PROGRAM Fixture1_Auto
VAR
	
nState_Door    : INT; // 0: Idle, 10: Starting, 20: Rotating, 30: Stopping
	
END_VAR




/////////////// OPERATOR LOAD PART FIX 1 ///////////////

		IF Memory_DB.M_Auto_Active AND 
		   Memory_DB.M_Power_On AND 
		   Inputs.i_Front_Door_Up
		   THEN   
		IF Memory_DB.M_FX1_LOAD1 AND Memory_DB.M_Turntable_POS1_Reached AND Memory_DB.M_Fixture1_TR_POS1_Reached  THEN
		  Inputs.i_FX1_PART_CONTROL_B1 := TRUE;
		  Inputs.i_FX1_PART_CONTROL_B2 := TRUE;
		  Inputs.i_FX1_PART_CONTROL_B3 := TRUE;
		  Inputs.i_FX1_PART_CONTROL_B4 := TRUE;
		  Inputs.i_FX1_PART_CONTROL_B5 := TRUE;
		  Inputs.i_FX1_PART_CONTROL_B6 := TRUE;
		  Inputs.i_FX1_PART_CONTROL_B7 := TRUE;
		  Memory_DB.M_FX1_LOAD1_COMPLETED :=TRUE;
		
		ELSIF Memory_DB.M_Auto_Active AND Memory_DB.M_Turntable_POS1_Reached AND Memory_DB.M_Fixture1_TR_POS2_Reached AND Memory_DB.M_FX1_LOAD2 THEN
		      Inputs.i_FX1_PART_CONTROL_B15 := TRUE;
		      Inputs.i_FX1_PART_CONTROL_B16 := TRUE;
		      Inputs.i_FX1_PART_CONTROL_B17 := TRUE;
		      Inputs.i_FX1_PART_CONTROL_B18 := TRUE;
		      Inputs.i_FX1_PART_CONTROL_B19 := TRUE;
		      Inputs.i_FX1_PART_CONTROL_B20 := TRUE;
		      Inputs.i_FX1_PART_CONTROL_B21 := TRUE;
		      Memory_DB.M_FX1_LOAD2_COMPLETED :=TRUE;
		
		ELSIF Memory_DB.M_FX1_LOAD1_COMPLETED AND Memory_DB.M_FX1_LOAD2_COMPLETED THEN
			
			  Memory_DB.M_Fixture1_TR_Start :=TRUE;
			
		END_IF;
		END_IF;
		 IF 
		   Memory_DB. M_FX1_All_Initialise THEN
		   Memory_DB.M_Turntable_Start := TRUE;
	       Memory_DB.M_Turntable_POS1_CMD := TRUE;
		   Memory_DB.M_Turntable_POS2_CMD := FALSE;
		   Memory_DB.M_Fixture1_TR_Start := TRUE;
	       Memory_DB.M_Fixture1_TR_POS1_CMD := TRUE;
		   Memory_DB.M_Fixture1_TR_POS2_CMD := FALSE;
		   Memory_DB.M_REAR_DOOR_DOWN := TRUE;
		   Memory_DB.M_REAR_DOOR_Up := FALSE;
		   
		 END_IF
//////////////////LODING SIDE DOOR & TRUNION CONTROL OPERATION/////////////////
IF  Memory_DB.M_Auto_Active AND Memory_DB.M_Safety_Ok AND Memory_DB.M_Power_On  THEN
	
CASE nState_Door  OF
    0: // Default Position1 of Door Open
	IF Memory_DB.M_Turntable_POS1_Reached AND Memory_DB.M_Fixture1_TR_POS1_Reached THEN      
		Memory_DB.M_FRONT_DOOR_Down	:=FALSE;
		Memory_DB.M_FRONT_DOOR_UP	:=TRUE;	
		Memory_DB.M_R03_MH_Goto_Drop2:=FALSE;
		nState_Door := 10;
     END_IF  
	 
    10: // 1st Load completed and Door Close Command
 
        IF Memory_DB.M_FX1_LOAD1_COMPLETED AND Memory_DB.M_FX1_Cycle_Start_PB AND Inputs.i_Front_Door_Up THEN
		Memory_DB.M_FRONT_DOOR_Down	:=TRUE;
		Memory_DB.M_FRONT_DOOR_UP	:=FALSE;

            nState_Door := 20; // Trunion Move
        END_IF
		       
    20: // Clamp Sequence at Trunion Pos1
 
        IF Inputs.i_Front_Door_Down AND Memory_DB.M_Fixture1_TR_POS1_Reached THEN
		Memory_DB.A_FX1_CC1_CLAMPING_UNIT1_3_WP:=TRUE;
		Memory_DB.A_FX1_CC3_CLAMPING_UNIT3_3_WP:=TRUE;
		Memory_DB.A_FX1_CC5_CLAMPING_UNIT5_1_WP:=TRUE;
		Memory_DB.A_FX1_CC1_CLAMPING_UNIT1_3_HP:=FALSE;
		Memory_DB.A_FX1_CC3_CLAMPING_UNIT3_3_HP:=FALSE;
		Memory_DB.A_FX1_CC5_CLAMPING_UNIT5_1_HP:=FALSE;		

         nState_Door := 30; // Error State
        END_IF	

        
    30: // Trunion move to Position 2 for 2nd Load
 
        IF Inputs.i_Front_Door_Down AND Inputs.i_FX1_CC1_Clamp_1_Sensor_WP AND 
		Inputs.i_FX1_CC3_Clamp_1_Sensor_WP AND Inputs.i_FX1_CC5_Clamp_1_Sensor_WP THEN
		Memory_DB.M_Fixture1_TR_POS2_CMD:=TRUE;
		Memory_DB.M_Fixture1_TR_POS1_CMD:=FALSE;

            nState_Door := 40; // Error State
        END_IF		
        
    40: // Door Open command for 2nd Load
 
        IF Memory_DB.M_Fixture1_TR_POS2_Reached AND Inputs.i_Front_Door_Down THEN
		Memory_DB.M_FRONT_DOOR_Down:=FALSE;
		Memory_DB.M_FRONT_DOOR_UP  :=TRUE;

            nState_Door := 50; // Error State
        END_IF	
        
    50: // 2nd Load completed on Trunion & Door Close Command
 
        IF Memory_DB.M_FX1_LOAD2_COMPLETED AND Memory_DB.M_FX1_Cycle_Start_PB AND Inputs.i_Front_Door_Up THEN
		Memory_DB.M_FRONT_DOOR_Down      :=TRUE;
		Memory_DB.M_FRONT_DOOR_Up        :=FALSE;

            nState_Door := 60; // Error State
        END_IF
		
    60: // Clamp Sequence at Trunion Pos1
 
        IF Inputs.i_Front_Door_Down AND Memory_DB.M_Fixture1_TR_POS2_Reached THEN
		Memory_DB.A_FX1_CC2_CLAMPING_UNIT2_3_WP:=TRUE;
		Memory_DB.A_FX1_CC4_CLAMPING_UNIT4_3_WP:=TRUE;
		Memory_DB.A_FX1_CC6_CLAMPING_UNIT6_1_WP:=TRUE;
		Memory_DB.A_FX1_CC2_CLAMPING_UNIT2_3_HP:=FALSE;
		Memory_DB.A_FX1_CC4_CLAMPING_UNIT4_3_HP:=FALSE;
		Memory_DB.A_FX1_CC6_CLAMPING_UNIT6_1_HP:=FALSE;	

         nState_Door := 70; // Error State
        END_IF		
        
    70: // Move Trunion to Default/Pos1
 
        IF Memory_DB.M_Fixture1_TR_Start AND Inputs.i_Front_Door_Down AND Memory_DB.M_Fixture1_TR_POS2_Reached AND
		 Inputs.i_FX1_CC2_Clamp_1_Sensor_WP AND Inputs.i_FX1_CC4_Clamp_1_Sensor_WP AND Inputs.i_FX1_CC6_Clamp_1_Sensor_WP THEN
		Memory_DB.M_Fixture1_TR_POS1_CMD:=TRUE;
		Memory_DB.M_Fixture1_TR_POS2_CMD:=FALSE;

            nState_Door := 80; // Error State
        END_IF
		
    80: // Move TT Work position/Pos2
 
        IF Memory_DB.M_FX1_LOAD1_COMPLETED AND Memory_DB.M_FX1_LOAD2_COMPLETED AND Inputs.i_Front_Door_Down AND Memory_DB.M_Fixture1_TR_POS1_Reached AND Memory_DB.M_Turntable_POS1_Reached 
           AND Inputs.i_Rear_Door_Down AND Inputs.i_FX1_CC2_Clamp_1_Sensor_WP AND Inputs.i_FX1_CC4_Clamp_1_Sensor_WP AND Inputs.i_FX1_CC6_Clamp_1_Sensor_WP 
           AND Memory_DB.M_R01_Home AND Memory_DB.M_R02_Home AND Memory_DB.M_R03_MH_AtHome THEN
		   Memory_DB.M_Turntable_Start:=TRUE;
		   Memory_DB.M_Turntable_POS2_CMD :=TRUE;
		   Memory_DB.M_Turntable_POS1_CMD :=FALSE;
           Memory_DB.M_FRONT_DOOR_Down    :=FALSE;
		   
            nState_Door := 90; // Error State
        END_IF		

	90: // Robot Weld CMD for First Weld
 
       IF  Memory_DB.M_Fixture1_TR_POS1_Reached AND Memory_DB.M_Turntable_POS2_Reached 
           AND Inputs.i_Rear_Door_Down AND Inputs.i_FX1_CC2_Clamp_1_Sensor_WP AND Inputs.i_FX1_CC4_Clamp_1_Sensor_WP AND Inputs.i_FX1_CC6_Clamp_1_Sensor_WP 
           AND Memory_DB.M_R01_Home AND Memory_DB.M_R02_Home AND Memory_DB.M_R03_MH_AtHome THEN
		   Memory_DB.M_R01_Weld_Start:=TRUE;
		   Memory_DB.M_R02_Weld_Start:=TRUE;
		  
            nState_Door := 100; // Error State
      	END_IF			
		
	100: // Trunnion move to POS2 for second Weld
 
        IF Memory_DB.M_R01_Job_Done1 AND Memory_DB.M_R02_Job_Done1 AND Inputs.i_Rear_Door_Down AND Memory_DB.M_Fixture1_TR_POS1_Reached AND Memory_DB.M_Turntable_POS2_Reached AND Inputs.i_FX1_CC2_Clamp_1_Sensor_WP AND Inputs.i_FX1_CC4_Clamp_1_Sensor_WP AND Inputs.i_FX1_CC6_Clamp_1_Sensor_WP THEN
		   Memory_DB.M_Fixture1_TR_POS1_CMD:=FALSE;
		   Memory_DB.M_Fixture1_TR_POS2_CMD:=TRUE;
		  

            nState_Door := 110; // Error State
        END_IF				
		
		
	110: // Robot Weld CMD for Second Weld
 
        IF  Inputs.i_Rear_Door_Down AND Memory_DB.M_Fixture1_TR_POS2_Reached  AND Memory_DB.M_Turntable_POS2_Reached  
           AND Inputs.i_FX1_CC2_Clamp_1_Sensor_WP AND Inputs.i_FX1_CC4_Clamp_1_Sensor_WP AND Inputs.i_FX1_CC6_Clamp_1_Sensor_WP THEN
		   Memory_DB.M_R01_Weld_Start:=TRUE;
		   Memory_DB.M_R02_Weld_Start:=TRUE;
		  
            nState_Door := 120; // Error State
        END_IF					
		
		
	120: // Trunnion move to POS1 for Unload part
 
        IF Memory_DB.M_R01_Job_Done1 AND Memory_DB.M_R02_Job_Done1 AND Memory_DB.M_R01_Job_Done2 AND Memory_DB.M_R02_Job_Done2 AND Inputs.i_Rear_Door_Down AND Memory_DB.M_Fixture1_TR_POS2_Reached AND Memory_DB.M_Turntable_POS2_Reached AND Inputs.i_FX1_CC2_Clamp_1_Sensor_WP AND Inputs.i_FX1_CC4_Clamp_1_Sensor_WP AND Inputs.i_FX1_CC6_Clamp_1_Sensor_WP THEN
		   Memory_DB.M_Fixture1_TR_POS2_CMD :=FALSE;
		   Memory_DB.M_Fixture1_TR_POS1_CMD :=TRUE;
		   Memory_DB.M_R01_Weld_Start:=FALSE;
		   Memory_DB.M_R02_Weld_Start:=FALSE;
		   
            nState_Door := 130; // Error State
        END_IF					
		
			
	130: // Rear Door Open
 
        IF  Inputs.i_Rear_Door_Down AND Memory_DB.M_Fixture1_TR_POS1_Reached AND Memory_DB.M_Turntable_POS2_Reached AND Inputs.i_FX1_CC2_Clamp_1_Sensor_WP AND Inputs.i_FX1_CC4_Clamp_1_Sensor_WP AND Inputs.i_FX1_CC6_Clamp_1_Sensor_WP THEN
		   Memory_DB.M_Rear_DOOR_Up      :=TRUE;
		   Memory_DB.M_Rear_DOOR_Down    :=FALSE;
		  
		   
            nState_Door := 140; // Error State
        END_IF
	
		
	140: // MH Robot Part Unload Command
 
        IF Inputs.i_Rear_Door_Up AND Memory_DB.M_Fixture1_TR_POS1_Reached AND Memory_DB.M_Turntable_POS2_Reached AND Inputs.i_FX1_CC2_Clamp_1_Sensor_WP AND Inputs.i_FX1_CC4_Clamp_1_Sensor_WP AND Inputs.i_FX1_CC6_Clamp_1_Sensor_WP THEN
		   Memory_DB.M_R03_MH_Cycle_Start   :=TRUE;
		   Memory_DB.M_R03_MH_MovePounce    :=TRUE;
		  
		   
            nState_Door := 150; // Error State
        END_IF
	
	150: // MH Robot At Pounce and Fixture Clamp Open
 
     IF Memory_DB.M_R03_MH_MovePounce AND Inputs.i_Rear_Door_Up AND Memory_DB.M_Fixture1_TR_POS1_Reached AND Memory_DB.M_Turntable_POS2_Reached AND Inputs.i_FX1_CC1_Clamp_1_Sensor_WP AND Inputs.i_FX1_CC3_Clamp_1_Sensor_WP AND Inputs.i_FX1_CC5_Clamp_1_Sensor_WP THEN
		Memory_DB.A_FX1_CC1_CLAMPING_UNIT1_3_HP:=TRUE;
		Memory_DB.A_FX1_CC3_CLAMPING_UNIT3_3_HP:=TRUE;
		Memory_DB.A_FX1_CC5_CLAMPING_UNIT5_1_HP:=TRUE;
		Memory_DB.A_FX1_CC1_CLAMPING_UNIT1_3_WP:=FALSE;
		Memory_DB.A_FX1_CC3_CLAMPING_UNIT3_3_WP:=FALSE;
		Memory_DB.A_FX1_CC5_CLAMPING_UNIT5_1_WP:=FALSE;	
		  
		   
            nState_Door := 160; // Error State
     END_IF
	 
	 
	160: // MH Robot Part Pick1 Command
 
        IF Inputs.i_Rear_Door_Up AND Memory_DB.M_Fixture1_TR_POS1_Reached AND Memory_DB.M_Turntable_POS2_Reached AND Inputs.i_FX1_CC1_Clamp_1_Sensor_HP AND Inputs.i_FX1_CC3_Clamp_1_Sensor_HP AND Inputs.i_FX1_CC5_Clamp_1_Sensor_HP THEN
		   Memory_DB.M_R03_MH_Cycle_Start   :=FALSE;
		   Memory_DB.M_R03_MH_MovePounce    :=FALSE;
		  Memory_DB.M_R03_MH_Goto_Pick1     :=TRUE;
		  Inputs.i_FX1_PART_CONTROL_B1 := FALSE;
		  Inputs.i_FX1_PART_CONTROL_B2 := FALSE;
		  Inputs.i_FX1_PART_CONTROL_B3 := FALSE;
		  Inputs.i_FX1_PART_CONTROL_B4 := FALSE;
		  Inputs.i_FX1_PART_CONTROL_B5 := FALSE;
		  Inputs.i_FX1_PART_CONTROL_B6 := FALSE;
		  Inputs.i_FX1_PART_CONTROL_B7 := FALSE;
		   
            nState_Door := 170; // Error State
        END_IF	
		
		
	170: // MH Robot Move to Paunce 
 
        IF Inputs.i_Rear_Door_Up AND Memory_DB.M_Fixture1_TR_POS1_Reached AND Memory_DB.M_Turntable_POS2_Reached AND Inputs.i_FX1_CC2_Clamp_1_Sensor_WP AND Inputs.i_FX1_CC4_Clamp_1_Sensor_WP AND Inputs.i_FX1_CC6_Clamp_1_Sensor_WP THEN
		  
		   Memory_DB.M_R03_MH_MovePounce    :=TRUE;	  
		   
            nState_Door := 180; // Error State
        END_IF		
		
	180: // Trunion rotate to Pos2
 
        IF Inputs.i_Rear_Door_Up AND Memory_DB.M_R03_MH_Pick1_Done AND Memory_DB.M_Fixture1_TR_POS1_Reached AND Memory_DB.M_Turntable_POS2_Reached AND Inputs.i_FX1_CC2_Clamp_1_Sensor_WP AND Inputs.i_FX1_CC4_Clamp_1_Sensor_WP AND Inputs.i_FX1_CC6_Clamp_1_Sensor_WP THEN
		   Memory_DB.M_Fixture1_TR_POS1_CMD:=FALSE;
		   Memory_DB.M_Fixture1_TR_POS2_CMD:=TRUE;
		    		   
            nState_Door := 190; // Error State
        END_IF		
			
	190: // Fixture clamp Open
 
       IF Inputs.i_Rear_Door_Up AND Memory_DB.M_R03_MH_Pick1_Done AND Memory_DB.M_Fixture1_TR_POS2_Reached AND Memory_DB.M_Turntable_POS2_Reached AND Inputs.i_FX1_CC2_Clamp_1_Sensor_WP AND Inputs.i_FX1_CC4_Clamp_1_Sensor_WP AND Inputs.i_FX1_CC6_Clamp_1_Sensor_WP THEN
		Memory_DB.A_FX1_CC2_CLAMPING_UNIT2_3_HP:=TRUE;
		Memory_DB.A_FX1_CC4_CLAMPING_UNIT4_3_HP:=TRUE;
		Memory_DB.A_FX1_CC6_CLAMPING_UNIT6_1_HP:=TRUE;
		Memory_DB.A_FX1_CC2_CLAMPING_UNIT2_3_WP:=FALSE;
		Memory_DB.A_FX1_CC4_CLAMPING_UNIT4_3_WP:=FALSE;
		Memory_DB.A_FX1_CC6_CLAMPING_UNIT6_1_WP:=FALSE;	
		    		   
            nState_Door := 200; // Error State
       END_IF			
		
	  200: // MH Robot Part Pick2 Command
 
       IF Inputs.i_Rear_Door_Up AND Memory_DB.M_R03_MH_Pick1_Done AND Memory_DB.M_Fixture1_TR_POS2_Reached AND Memory_DB.M_Turntable_POS2_Reached AND Inputs.i_FX1_CC2_Clamp_1_Sensor_HP AND Inputs.i_FX1_CC4_Clamp_1_Sensor_HP AND Inputs.i_FX1_CC6_Clamp_1_Sensor_HP THEN
		  Memory_DB.M_R03_MH_MovePounce    :=FALSE;
		  Memory_DB.M_R03_MH_Goto_Pick2     :=TRUE;
		  Inputs.i_FX1_PART_CONTROL_B15 := FALSE;
		  Inputs.i_FX1_PART_CONTROL_B16 := FALSE;
		  Inputs.i_FX1_PART_CONTROL_B17 := FALSE;
		  Inputs.i_FX1_PART_CONTROL_B18 := FALSE;
		  Inputs.i_FX1_PART_CONTROL_B19 := FALSE;
		  Inputs.i_FX1_PART_CONTROL_B20 := FALSE;
		  Inputs.i_FX1_PART_CONTROL_B21 := FALSE;
		    		   
            nState_Door := 210; // Error State
       END_IF	
 
	 210: // Trunion rotate to POS1  
	   IF Inputs.i_Rear_Door_Up AND Memory_DB.M_R03_MH_Pick1_Done AND Memory_DB.M_Fixture1_TR_POS2_Reached AND Memory_DB.M_Turntable_POS2_Reached AND Inputs.i_FX1_CC2_Clamp_1_Sensor_HP AND Inputs.i_FX1_CC4_Clamp_1_Sensor_HP AND Inputs.i_FX1_CC6_Clamp_1_Sensor_HP THEN
		  Memory_DB.M_Fixture1_TR_POS1_CMD := TRUE;
		  Memory_DB.M_Fixture1_TR_POS2_CMD := FALSE; 
		  
		    		   
            nState_Door := 220; // Error State
       END_IF	 
	   
	 220: // Rear Door Down
 
       IF Inputs.i_Rear_Door_Up AND Memory_DB.M_R03_MH_Pick1_Done AND Memory_DB.M_R03_MH_Pick2_Done AND Memory_DB.M_Fixture1_TR_POS1_Reached AND Memory_DB.M_Turntable_POS2_Reached THEN
		   Memory_DB.M_Rear_DOOR_Down   :=TRUE;
		   Memory_DB.M_Rear_DOOR_Up     :=FALSE;
		  Memory_DB.M_R03_MH_MovePounce :=TRUE;
		  Memory_DB.M_R01_Job_Done1     :=FALSE;   
		  Memory_DB.M_R01_Job_Done2     :=FALSE;    
          Memory_DB.M_R02_Job_Done1     :=FALSE;  
		  Memory_DB.M_R02_Job_Done2     :=FALSE;   
          Memory_DB.M_R03_MH_Goto_Pick1 :=FALSE; 
		  Memory_DB.M_R03_MH_Goto_Pick2 :=FALSE;
            nState_Door := 230; // Error State
       END_IF	
 	
	
	    230: // Robot Go to Drop1 & Drop2
 
       IF Inputs.i_Rear_Door_Down AND Memory_DB.M_R03_MH_Pick1_Done AND Memory_DB.M_R03_MH_Pick2_Done AND Memory_DB.M_Fixture1_TR_POS1_Reached AND Memory_DB.M_Turntable_POS2_Reached THEN
		  
		  Memory_DB.M_R03_MH_Goto_Drop1 :=TRUE;	    
		  Memory_DB.M_R03_MH_MovePounce :=FALSE;  
		   
 
            nState_Door := 240; // Error State
       END_IF
	
	   240: // Robot Go to Drop2 
 
       IF Inputs.i_Rear_Door_Down AND Memory_DB.M_R03_MH_Pick1_Done AND Memory_DB.M_R03_MH_Pick2_Done AND Memory_DB.M_Fixture1_TR_POS1_Reached AND Memory_DB.M_Turntable_POS2_Reached THEN
		  
		  Memory_DB.M_R03_MH_Goto_Drop1 :=FALSE;
		  Memory_DB.M_R03_MH_Goto_Drop2  :=TRUE;   
		  Memory_DB.M_R03_MH_MovePounce :=FALSE;  
		  
 
            nState_Door := 250; // Error State
       END_IF

	 250: // TT Rotate to load position 
 
       IF Memory_DB.M_Fixture1_TR_POS1_Reached AND Memory_DB.M_Turntable_POS1_Reached THEN
		  	   
 
            nState_Door := 0; // Error State
       END_IF
END_CASE;
END_IF;

END_PROGRAM

(* stored: Version 1.1.0.1, ProductVersion 3.1.4024.16
   POU Fixture1_Auto: Id {bd9c96be-cb9d-4e25-b345-dbf5d3a724a5}, SpecialFunc None *)
